/// calibration that is determined by calibration sequences of the unit (static offsets, shifts)
TYPE XyTableDataCalibration :
STRUCT
END_STRUCT
END_TYPE

(* stored: Version 1.1.0.1
   DUT XyTableDataCalibration: Id {acb590e8-e3ba-42a1-9be4-ea6312f15084} *)
